{attribute 'qualified_only'}
VAR_GLOBAL
	sPistonEndStopMessages : STRING;
END_VAR

(* stored: Version 1.1.0.1, ProductVersion 3.1.4024.10
   GVL HMI: Id {f4505ebe-755d-4b1a-9777-bfeb2aca0966} *)
